FUNCTION_BLOCK Test_Raises_OnHoursChanged EXTENDS TUnitTestBase
IMPLEMENTS 
    IEventHandler_OnHourChanged
VAR
    NowFromEvent : TIMESTRUCT;
    
    OnHoursChanged_Raised    : BOOL;
END_VAR

METHOD  Execute
VAR_INST
    ClockEventSource : TClockEventSource;
    Now              : TIMESTRUCT := (wDay := 23, wMonth := 12, wYear := 1945, wHour := 22, wMinute := 20, wSecond := 18);
    OneHourLater     : TIMESTRUCT := (wDay := 23, wMonth := 12, wYear := 1945, wHour := 23, wMinute := 20, wSecond := 18);
END_VAR
OnHoursChanged_Raised := FALSE;

ClockEventSource.Event_HoursChanged.ClearEventHandlers().AddEventHandler(THIS^);

ClockEventSource.Init(Now := Now);
ClockEventSource(Now := OneHourLater);

Assertion.AssertEquals_BOOL(
    Expected := TRUE,
    Actual   := OnHoursChanged_Raised,
    ObjectName := _TestName,
    VariableName  := 'OnHoursChanged_Raised');

Assertion.AssertEquals_STRUCT(
    Expected := OneHourLater,
    Actual   := NowFromEvent,
    ObjectName := _TestName,
    VariableName  := 'NowFromEvent');

Test_Finished();
END_METHOD

METHOD OnHourChanged
VAR_INPUT
	Now	: Tc2_Utilities.TIMESTRUCT;
END_VAR
NowFromEvent := Now;
OnHoursChanged_Raised := TRUE;
END_METHOD

END_FUNCTION_BLOCK

(* stored: Version 1.1.0.1, ProductVersion 3.1.4024.3
   POU Test_Raises_OnHoursChanged: Id {e535cbdc-dab6-0b06-08b5-ae85ab52fd8c}, SpecialFunc None
   Method Execute: Id {7138b20d-681b-0e17-0c54-b120fc243fda}
   Method OnHourChanged: Id {a7186963-839c-0647-0738-9ed23cb7af23} *)
